Yaskawa INFORM job: output.JBI

/JOB
//NAME output
//POS
///NPOS 42,0,0,0,0,0
///TOOL 0
///POSTYPE PULSE
///PULSE
C00000=0,0,0,0,0,0
C00001=-30979, 23934, -39608, 0, 38368, 12013
C00002=-12793, 15670, -47360, 0, 39276, 4961
C00003=-16213, -10378, -68048, 0, 39663, 6287
C00004=-16112, -10408, -68069, 0, 39661, 6248
C00005=-12712, 15650, -47379, 0, 39277, 4929
C00006=6931, 14527, -48388, 0, 39372, -2688
C00007=8819, -12085, -69202, 0, 39555, -3420
C00008=8923, -12068, -69191, 0, 39556, -3460
C00009=7013, 14539, -48378, 0, 39371, -2719
C00010=25796, 20793, -42620, 0, 38756, -10003
C00011=32155, -3011, -62784, 0, 39941, -12469
C00012=35604, -687, -61028, 0, 39965, -13806
C00013=25449, 36985, -26287, 0, 36221, -9868
C00014=28015, 38595, -24558, 0, 35899, -10863
C00015=21755, 77972, 22596, 0, 24824, -8436
C00016=19699, 76456, 20633, 0, 25348, -7639
C00017=25426, 37097, -26168, 0, 36199, -9860
C00018=27990, 38706, -24438, 0, 35877, -10854
C00019=12701, 94342, 44380, 0, 18779, -4925
C00020=13945, 73298, 16578, 0, 26417, -5407
C00021=21740, 78109, 22774, 0, 24776, -8430
C00022=5269, 91294, 40247, 0, 19956, -2043
C00023=5794, 70690, 13263, 0, 27277, -2247
C00024=13891, 73273, 16546, 0, 26425, -5387
C00025=12652, 94313, 44340, 0, 18790, -4906
C00026=-2263, 90797, 39576, 0, 20145, 877
C00027=-2489, 70258, 12716, 0, 27418, 965
C00028=5739, 70680, 13250, 0, 27281, -2225
C00029=5219, 91283, 40231, 0, 19960, -2024
C00030=-9751, 92805, 42291, 0, 19375, 3781
C00031=-10715, 71992, 14914, 0, 26850, 4155
C00032=-2544, 70262, 12721, 0, 27417, 987
C00033=-2313, 90802, 39583, 0, 20143, 897
C00034=-30949, 24045, -39501, 0, 38353, 12001
C00035=-15971, 16709, -46416, 0, 39182, 6193
C00036=-9801, 92827, 42321, 0, 19367, 3800
C00037=-15892, 16684, -46439, 0, 39184, 6162
C00038=-10877, 69206, 11390, 0, 27758, 4218
C00039=19712, 73586, 16946, 0, 26321, -7644
C00040=28320, 22367, -41121, 0, 38568, -10982
C00041=-15892, 16684, -46439, 0, 39184, 6162
//INST
///DATE 2015/05/11 9:31
///ATTR SC,RW
///GROUP1 RB1
NOP
MOVJ C00000 VJ=5
MOVJ C00001 VJ=5
MOVL C00002 V=100
MOVL C00003 V=100
MOVJ C00004 VJ=5
MOVL C00005 V=100
MOVL C00006 V=100
MOVL C00007 V=100
MOVJ C00008 VJ=5
MOVL C00009 V=100
MOVL C00010 V=100
MOVL C00011 V=100
MOVJ C00012 VJ=5
MOVL C00013 V=100
MOVL C00014 V=100
MOVJ C00015 VJ=5
MOVL C00016 V=100
MOVL C00017 V=100
MOVL C00018 V=100
MOVJ C00019 VJ=5
MOVL C00020 V=100
MOVL C00021 V=100
MOVJ C00022 VJ=5
MOVL C00023 V=100
MOVL C00024 V=100
MOVL C00025 V=100
MOVJ C00026 VJ=5
MOVL C00027 V=100
MOVL C00028 V=100
MOVL C00029 V=100
MOVJ C00030 VJ=5
MOVL C00031 V=100
MOVL C00032 V=100
MOVL C00033 V=100
MOVJ C00034 VJ=5
MOVL C00035 V=100
MOVL C00036 V=100
MOVJ C00037 VJ=5
MOVL C00038 V=100
MOVL C00039 V=100
MOVL C00040 V=100
MOVL C00041 V=100
MOVJ C00000 VJ=5
END
